FUNCTION_BLOCK FB_BottleFillingMachine IMPLEMENTS I_Machine


VAR
	eState : E_MachineState;
    eMode  : E_MachineMode;
	
	fbConveyor      : FB_Conveyor;
    fbFillingUnit   : FB_FillingUnit;
    fbBottleCounter : FB_BottleCounter;
	
	tConveyerTime : TIME := T#5S;
	tFillingTime : TIME := T#3S;
	

	tonSimBottle : TON;
    tonSimLevel  : TON;

END_VAR

METHOD Execute
IF GVL_IO.g_bStopButton THEN
	GVL_IO.g_bAlarmLamp := TRUE;
    eState := E_MachineState.Stopped;
END_IF

IF GVL_IO.g_bresetCounter THEN 
	fbBottleCounter.Reset();
	GVL_IO.g_bresetCounter := FALSE;
END_IF

IF GVL_IO.g_bBottleSensor AND GVL_IO.g_bLevelSensor THEN
	GVL_IO.g_bAlarmLamp := TRUE;
	eState := E_MachineState.stopped;
	GVL_IO.g_sStatusofMachine := 'Error';	
END_IF

CASE eState OF

    E_MachineState.Idle:
			GVL_IO.g_eState := E_MachineState.Idle;
			fbConveyor.stop();
			fbFillingUnit.StopFill();
			start();
			
    E_MachineState.Running:
		IF emode = E_MachineMode.none THEN 
			GVL_IO.g_sStatusofMachine := 'Select any Mode';
		ELSE
			GVL_IO.g_sStatusofMachine := 'Bottle is Moving';
			GVL_IO.g_conveyorStatus := 'conveyor is running';
			IF (emode = E_MachineMode.auto) THEN 
					GVL_IO.g_bSIM_BottleSensor := FALSE;
					fbConveyor.start();
					tonSimBottle(IN := NOT GVL_IO.g_bSIM_BottleSensor, PT := tConveyerTime);
					
					IF tonSimBottle.Q THEN 
						GVL_IO.g_bSIM_BottleSensor := TRUE;
						GVL_IO.g_eState := E_MachineState.Running;
					END_IF
					
					IF GVL_IO.g_bBottleSensor OR GVL_IO.g_bSIM_BottleSensor THEN 
						fbConveyor.stop();
						tonSimBottle(IN := FALSE);
						eState := E_MachineState.Filling;
					END_IF
					
					IF tonSimBottle.Q AND NOT (GVL_IO.g_bBottleSensor OR GVL_IO.g_bSIM_BottleSensor) THEN		
						GVL_IO.g_bAlarmLamp := TRUE;			
						eState := E_MachineState.Stopped;		
					END_IF
					
			ELSE
				IF GVL_IO.g_bBottleSensor THEN 
					GVL_IO.g_sStatusofMachine := 'Bottle detected';
					GVL_IO.g_conveyorStatus := 'conveyor is stopped';
					eState := E_MachineState.Filling;			
				END_IF
			END_IF
		END_IF
		
			

    E_MachineState.Filling:
			GVL_IO.g_sStatusofMachine := 'Bottle detected and filling started';
			GVL_IO.g_conveyorStatus := 'Conveyor is stopped';
			IF (emode = E_MachineMode.auto) THEN		
				GVL_IO.g_bSIM_LevelSensor := FALSE;
				fbFillingUnit.StartFill();
				
				tonSimLevel(IN := NOT GVL_IO.g_bSIM_LevelSensor, PT := tFillingTime);
				
				IF tonSimLevel.Q THEN 
					GVL_IO.g_sStatusofMachine := 'Filling Completed';
					GVL_IO.g_bSIM_LevelSensor := TRUE;
					GVL_IO.g_eState := E_MachineState.Filling;
				END_IF
				
				IF GVL_IO.g_bLevelSensor OR GVL_IO.g_bSIM_LevelSensor THEN 
					fbFillingUnit.StopFill();
					tonSimLevel(IN := FALSE);
					
					eState := E_MachineState.Running;
					fbBottleCounter.BottleCount();			
				END_IF
				
				IF tonSimLevel.Q AND NOT (GVL_IO.g_bLevelSensor OR GVL_IO.g_bSIM_LevelSensor) THEN
					GVL_IO.g_bAlarmLamp := TRUE;		
					eState := E_MachineState.Stopped;
				END_IF
			ELSE
				IF GVL_IO.g_bLevelSensor THEN 
					eState := E_MachineState.stopped;
					fbBottleCounter.BottleCount();
					GVL_IO.g_sStatusofMachine := 'Filling Completed';
				END_IF
			END_IF
			

    E_MachineState.Stopped:
			stop();
			GVL_IO.g_conveyorStatus := 'Conveyor is stopped';
			GVL_IO.g_sStatusofMachine := 'Process Completed';
			fbConveyor.Stop();
			fbFillingUnit.StopFill();
			


END_CASE;
END_METHOD

METHOD SelectMode : E_MachineMode
VAR_INPUT
	eSelectedMode : E_MachineMode;
END_VAR
eMode := eSelectedMode;
END_METHOD

{warning 'add method implementation '}
METHOD Start
IF GVL_IO.g_bStartButton THEN
	GVL_IO.g_bAlarmLamp := FALSE;
    eState := E_MachineState.Running;
END_IF
END_METHOD

{warning 'add method implementation '}
METHOD Stop
IF GVL_IO.g_bStopButton THEN
    eState := E_MachineState.Stopped;
END_IF
END_METHOD

END_FUNCTION_BLOCK

(* stored: Version 1.1.0.1, ProductVersion 3.1.4024.16
   POU FB_BottleFillingMachine: Id {8b303d4f-0cdf-4b38-8abc-9572eb954d2c}, SpecialFunc None
   Method Execute: Id {fe08e00b-04d9-496e-9e8b-964636ee76f3}
   Method SelectMode: Id {af7a7f0c-87c3-420e-803b-4cfcacfc6a80}
   Method Start: Id {16419386-e6e4-48f4-b76c-871cca0c0b49}
   Method Stop: Id {848cb335-2e76-42e0-bb57-9e9f71afbe6e} *)
